//The Edge Counter 1Ch counts the amount of raised events. An event is raised when the signal of the input channel passes the configured edge at a specific threshold. Optional a boolean signal for Enable Execution can be selected, so that the algorithm is just active if the value of the selected signal is TRUE.
FUNCTION_BLOCK FB_N3_M3_EdgeCounter1Ch
VAR_INPUT
	fDataIn: LREAL; 
	tTimestamp: ULINT; 
	bEnableExecution: BOOL := TRUE; 
	bReset: BOOL; 
	bReconfigure: BOOL := TRUE;
END_VAR
VAR_INPUT PERSISTENT
	stThresholdEdge: ST_ALY_Threshold; 
	fTolerance: LREAL; 
END_VAR
VAR_OUTPUT
	bError: BOOL;
	ipTcResult: I_TcMessage;
	bNewResult: BOOL;
	bEdge: BOOL;
	nCount: ULINT;
	fbTimeLastEvent: FB_ALY_DateTime;
END_VAR
VAR
	
	R_TRIG_Reconfigure: R_TRIG;
	
	fbALY_EdgeCounter_1Ch: FB_ALY_EdgeCounter_1Ch := ( bPersistent:= TRUE );
END_VAR
VAR PERSISTENT
	bConfigured: BOOL;
END_VAR

METHOD Call : BOOL
VAR_INPUT
	nCurrentContext: DWORD;
END_VAR
VAR
END_VAR
IF NOT bConfigured THEN
	bConfigured:= TRUE;

	fTolerance:= 0;

	stThresholdEdge.eComparisonOperator:= E_ALY_ComparisonOperator.GreaterThanOrEqualTo;
	stThresholdEdge.fThreshold:= 1;

	fbALY_EdgeCounter_1Ch.fTolerance:= fTolerance;
END_IF

R_TRIG_Reconfigure(CLK:= bReconfigure);
IF R_TRIG_Reconfigure.Q THEN
	fbALY_EdgeCounter_1Ch.ConfigureChannel(stThresholdEdge:= stThresholdEdge);

	fbALY_EdgeCounter_1Ch.Configure();

	bReconfigure:= FALSE;
END_IF

IF bReset THEN
	Reset();
END_IF

IF bEnableExecution THEN
	IF F_HasContext(nCurrentContext, nContext) THEN
		fbALY_EdgeCounter_1Ch.SetChannelValue(Input:= fDataIn);

		fbALY_EdgeCounter_1Ch.Call(tTimestamp:= tTimestamp);

		bNewResult:= fbALY_EdgeCounter_1Ch.bNewResult;
		bEdge:= fbALY_EdgeCounter_1Ch.bEdge;
		nCount:= fbALY_EdgeCounter_1Ch.nCount;
		fbTimeLastEvent:= fbALY_EdgeCounter_1Ch.fbTimeLastEvent;

		bError:= fbALY_EdgeCounter_1Ch.bError;
		ipTcResult:= fbALY_EdgeCounter_1Ch.ipResultMessage;
	END_IF
ELSE
	bNewResult:= FALSE;
END_IF
END_METHOD

METHOD Reset : BOOL
VAR
END_VAR
Reset:= fbALY_EdgeCounter_1Ch.Reset();

bNewResult:= fbALY_EdgeCounter_1Ch.bNewResult;
bEdge:= fbALY_EdgeCounter_1Ch.bEdge;
nCount:= fbALY_EdgeCounter_1Ch.nCount;
fbTimeLastEvent:= fbALY_EdgeCounter_1Ch.fbTimeLastEvent;

bError:= NOT Reset;
ipTcResult:= fbALY_EdgeCounter_1Ch.ipResultMessage;
END_METHOD

PROPERTY nContext : DWORD
GET
nContext:= E_VirtualInput.eContext_V1_Virtual_Input_Source;
END_GET
END_PROPERTY

END_FUNCTION_BLOCK

(* stored: POU FB_N3_M3_EdgeCounter1Ch: Id ed0f5008-9824-4010-b6b1-f0f848ff5fa8, SpecialFunc None
   Method Call: Id abb5f69c-5d25-4c04-9b6a-ab4551c60460
   Method Reset: Id 43f90699-3c38-4e85-9559-bda03e68c1c6
   Property nContext: Id 30b1c897-0bde-4a1d-b10f-8ee58b36f5bf
   Get Get: Id 5de59ced-aff0-4275-ad9d-f161d4743c2b *)
